{attribute 'qualified_only'}
VAR_GLOBAL
//Input to PLC from process
	ixAGVStrobe		AT %I*:	BOOL;	(* AGV strobe signal *)
	iiAtPos			AT %I*:	INT;	(* Actual position of AGV *)
	
//Output from PLC to process
	qxPLCStrobe		AT %Q*:	BOOL;	(* PLC strobe signal *)
	qiGotoPos		AT %Q*:	INT;	(* Target position for AGV *)
	
	sTargetList : ARRAY [1..5] OF STRING := ['HOME','A', 'B', 'C', 'D'];
	Position : INT:=0;
	ixStartButton : BOOL;
	ixStopButton : BOOL;
	ixResetButton : BOOL;
	qxDIsplay_Pos : STRING;
	qxReadylamp : BOOL;
	qxMovinglamp : BOOL;
	qxStoplamp : BOOL;
	qxStopEvent : BOOL;
END_VAR

(* stored: Version 1.1.0.1, ProductVersion 3.1.4024.12
   GVL GVL: Id {816111f0-16ef-4f4d-a70e-f3df38e5b1aa} *)
